// TwinCAT 3 PLC project Untitled1
// ProgramVersion: 3.1.4022.4
// libraries:
//   VisuElemBase, * (System)
//   VisuElems, * (System)
//   VisuElemsSpecialControls, * (System)
//   VisuElemsWinControls, * (System)
//   VisuInputs, * (System)
//   VisuNativeControl, * (System)
//   Tc2_FTP, * (Beckhoff Automation GmbH)
//   Tc2_MC2, * (Beckhoff Automation GmbH)
//   Tc2_NCI, * (Beckhoff Automation GmbH)
//   Tc2_Standard, * (Beckhoff Automation GmbH)
//   Tc2_System, * (Beckhoff Automation GmbH)
//   Tc2_Utilities, * (Beckhoff Automation GmbH)
//   Tc3_IotBase, * (Beckhoff Automation GmbH)
//   Tc3_JsonXml, * (Beckhoff Automation GmbH)
//   Tc3_Module, * (Beckhoff Automation GmbH)
//   VisuElemsDateTime Interfaces,newest,Intern
// project tree:
//   / GlobalTextList.TcGTLO, PlcTask.TcTTO, Visualization Manager.TcVMO (not stored)
//   GVLs/ COM.TcGVL, GVL.TcGVL
//   POUs/ ERROR.TcPOU, FTP.TcPOU, INIT.TcPOU, MAIN.TcPOU, POSITION.TcPOU, submqtt.TcPOU (not stored), commandDecoder.TcPOU
//   VISUs/ goPositionAbs.TcVIS, goPositionRel.TcVIS, Homing.TcVIS, Basic.TcVIS
// real-time tasks:
//   TASK PlcTask: cycle T#10ms, priority 20, ADS port 350
// motion (NC):
//   TASK NC-Task 1 SAF: cycle T#2ms, priority 4, ADS port 501
//   TASK NC-Task 1 SVB: cycle T#10ms, priority 8, ADS port 511
//   AXIS Axis X1 (id 1)
//     OtherSettings: AllowMotionCmdToSlave=true
//     encoder EncType=4
//       EncPara: ScaleFactorNumerator=40, ScaleFactorDenominator=12800, Inverse=true, MaxCount=#x0000ffff
//         SoftEndMinControl: Enable=true
//         SoftEndMaxControl: Enable=true, Range=275
//         Inc: RefSearchInverse=true, RefSyncInverse=false, RefMode=1, RefSoftSyncMask=#x0000ffff
//     drive DrvType=24
//       DrvPara: Inverse=true
//         Analog: VeloReferenz=400, ScaleFactorActTorque=0.1
//         TimeComp: TaskDelayCycles=1
//     controller CtrType=1
//       CtrPara: PriorControlFactor=1
//         PID: PosKp=25
//         Observer: BandWidth=20
//   AXIS Axis X2 (id 2)
//     OtherSettings: AllowMotionCmdToSlave=true
//     encoder EncType=4
//       EncPara: ScaleFactorNumerator=40, ScaleFactorDenominator=12800, Inverse=true, MaxCount=#x0000ffff
//         Inc: RefSoftSyncMask=#x0000ffff
//     drive DrvType=24
//       DrvPara: Inverse=true
//         Analog: VeloReferenz=400, ScaleFactorActTorque=0.1
//         TimeComp: TaskDelayCycles=1
//     controller CtrType=1
//       CtrPara: PriorControlFactor=1
//         PID: PosKp=25
//         Observer: BandWidth=20
//   AXIS Axis Y (id 4)
//     OtherSettings: AllowMotionCmdToSlave=true
//     encoder EncType=4
//       EncPara: ScaleFactorNumerator=40, ScaleFactorDenominator=12800, Inverse=true, MaxCount=#x0000ffff
//         SoftEndMinControl: Enable=true
//         SoftEndMaxControl: Enable=true, Range=275
//         Inc: RefSearchInverse=true, RefSyncInverse=false, RefMode=1, RefSoftSyncMask=#x0000ffff
//     drive DrvType=24
//       DrvPara: Inverse=true
//         Analog: VeloReferenz=400, ScaleFactorActTorque=0.1
//         TimeComp: TaskDelayCycles=1
//     controller CtrType=1
//       CtrPara: PriorControlFactor=1
//         PID: PosKp=25
//         Observer: BandWidth=20
//   AXIS Axis Z (id 3)
//     Velo: SlowManual=2, FastManual=5
//     OtherSettings: AllowMotionCmdToSlave=true
//     encoder EncType=4
//       EncPara: ScaleFactorNumerator=1, ScaleFactorDenominator=12800, MaxCount=#x0000ffff
//         Inc: RefSoftSyncMask=#x0000ffff
//     drive DrvType=24
//       Analog: VeloReferenz=10, ScaleFactorActTorque=0.1
//       TimeComp: TaskDelayCycles=1
//     controller CtrType=1
//       CtrPara: PriorControlFactor=1
//         PID: PosKp=25
//         Observer: BandWidth=20
// I/O:
//   DEVICE Device 3 (EtherCAT), AmsNetId 10.86.134.48.4.1
//     Term 1 (EK1100) [EK1100 EtherCAT Coupler (2A E-Bus)]
//       Term 2 (EL7031-0030) [EL7031-0030 1Ch. Stepper motor output stage (24V, 2.8A)]
//       Term 3 (EL7031-0030) [EL7031-0030 1Ch. Stepper motor output stage (24V, 2.8A)]
//       Term 4 (EL7031-0030) [EL7031-0030 1Ch. Stepper motor output stage (24V, 2.8A)]
//       Term 5 (EL7031-0030) [EL7031-0030 1Ch. Stepper motor output stage (24V, 2.8A)]
//       Term 6 (EL1008) [EL1008 8Ch. Dig. Input 24V, 3ms]
//       Term 7 (EL9011) [EL9011 End Terminal]
// variable links:
//   NC-Task 1 SAF/Axes/Axis X1 <-> Device 3 (EtherCAT)/Term 1 (EK1100)/Term 2 (EL7031-0030)
//     Drive/Inputs/In/nState1 @bit 3 <-> STM Status/Status/Error
//     Drive/Inputs/In/nState1 @bit 5 <-> STM Status/Status/Moving negative
//     Drive/Inputs/In/nState1 @bit 4 <-> STM Status/Status/Moving positive
//     Drive/Inputs/In/nState1 @bit 1 <-> STM Status/Status/Ready
//     Drive/Inputs/In/nState1 <-> STM Status/Status/Ready to enable
//     Drive/Inputs/In/nState1 @bit 6 <-> STM Status/Status/Torque reduced
//     Drive/Inputs/In/nState1 @bit 2 <-> STM Status/Status/Warning
//     Drive/Inputs/In/nState2 @bit 3 <-> STM Status/Status/Digital input 1
//     Drive/Inputs/In/nState2 @bit 4 <-> STM Status/Status/Digital input 2
//     Drive/Inputs/In/nState2 @bit 5 <-> STM Status/Status/Sync error
//     Drive/Inputs/In/nState2 @bit 7 <-> STM Status/Status/TxPDO Toggle
//     Drive/Inputs/In/nState4 @bit 1 <-> WcState/InputToggle
//     Drive/Inputs/In/nState4 <-> WcState/WcState
//     Drive/Outputs/Out/nCtrl1 <-> STM Control/Control/Enable
//     Drive/Outputs/Out/nCtrl1 @bit 2 <-> STM Control/Control/Reduce torque
//     Drive/Outputs/Out/nCtrl1 @bit 1 <-> STM Control/Control/Reset
//     Drive/Outputs/Out/nDataOut2[0] <-> STM Velocity/Velocity
//     Enc/Inputs/In/nDataIn1[0] <-> ENC Status compact/Counter value
//     Enc/Inputs/In/nDataIn2[0] <-> ENC Status compact/Latch value
//     Enc/Inputs/In/nState1 @bit 4 <-> ENC Status compact/Status/Counter overflow
//     Enc/Inputs/In/nState1 @bit 3 <-> ENC Status compact/Status/Counter underflow
//     Enc/Inputs/In/nState1 @bit 1 <-> ENC Status compact/Status/Latch extern valid
//     Enc/Inputs/In/nState1 @bit 2 <-> ENC Status compact/Status/Set counter done
//     Enc/Inputs/In/nState2 @bit 4 <-> ENC Status compact/Status/Status of extern latch
//     Enc/Inputs/In/nState2 @bit 5 <-> ENC Status compact/Status/Sync error
//     Enc/Inputs/In/nState2 @bit 7 <-> ENC Status compact/Status/TxPDO Toggle
//     Enc/Inputs/In/nState4 @bit 1 <-> WcState/InputToggle
//     Enc/Inputs/In/nState4 <-> WcState/WcState
//     Enc/Outputs/Out/nCtrl1 @bit 3 <-> ENC Control compact/Control/Enable latch extern on negative edge
//     Enc/Outputs/Out/nCtrl1 @bit 1 <-> ENC Control compact/Control/Enable latch extern on positive edge
//     Enc/Outputs/Out/nCtrl1 @bit 2 <-> ENC Control compact/Control/Set counter
//     Enc/Outputs/Out/nDataOut1[0] <-> ENC Control compact/Set counter value
//   NC-Task 1 SAF/Axes/Axis X2 <-> Device 3 (EtherCAT)/Term 1 (EK1100)/Term 3 (EL7031-0030)
//     Drive/Inputs/In/nState1 @bit 3 <-> STM Status/Status/Error
//     Drive/Inputs/In/nState1 @bit 5 <-> STM Status/Status/Moving negative
//     Drive/Inputs/In/nState1 @bit 4 <-> STM Status/Status/Moving positive
//     Drive/Inputs/In/nState1 @bit 1 <-> STM Status/Status/Ready
//     Drive/Inputs/In/nState1 <-> STM Status/Status/Ready to enable
//     Drive/Inputs/In/nState1 @bit 6 <-> STM Status/Status/Torque reduced
//     Drive/Inputs/In/nState1 @bit 2 <-> STM Status/Status/Warning
//     Drive/Inputs/In/nState2 @bit 3 <-> STM Status/Status/Digital input 1
//     Drive/Inputs/In/nState2 @bit 4 <-> STM Status/Status/Digital input 2
//     Drive/Inputs/In/nState2 @bit 5 <-> STM Status/Status/Sync error
//     Drive/Inputs/In/nState2 @bit 7 <-> STM Status/Status/TxPDO Toggle
//     Drive/Inputs/In/nState4 @bit 1 <-> WcState/InputToggle
//     Drive/Inputs/In/nState4 <-> WcState/WcState
//     Drive/Outputs/Out/nCtrl1 <-> STM Control/Control/Enable
//     Drive/Outputs/Out/nCtrl1 @bit 2 <-> STM Control/Control/Reduce torque
//     Drive/Outputs/Out/nCtrl1 @bit 1 <-> STM Control/Control/Reset
//     Drive/Outputs/Out/nDataOut2[0] <-> STM Velocity/Velocity
//     Enc/Inputs/In/nDataIn1[0] <-> ENC Status compact/Counter value
//     Enc/Inputs/In/nDataIn2[0] <-> ENC Status compact/Latch value
//     Enc/Inputs/In/nState1 @bit 4 <-> ENC Status compact/Status/Counter overflow
//     Enc/Inputs/In/nState1 @bit 3 <-> ENC Status compact/Status/Counter underflow
//     Enc/Inputs/In/nState1 @bit 1 <-> ENC Status compact/Status/Latch extern valid
//     Enc/Inputs/In/nState1 @bit 2 <-> ENC Status compact/Status/Set counter done
//     Enc/Inputs/In/nState2 @bit 4 <-> ENC Status compact/Status/Status of extern latch
//     Enc/Inputs/In/nState2 @bit 5 <-> ENC Status compact/Status/Sync error
//     Enc/Inputs/In/nState2 @bit 7 <-> ENC Status compact/Status/TxPDO Toggle
//     Enc/Inputs/In/nState4 @bit 1 <-> WcState/InputToggle
//     Enc/Inputs/In/nState4 <-> WcState/WcState
//     Enc/Outputs/Out/nCtrl1 @bit 3 <-> ENC Control compact/Control/Enable latch extern on negative edge
//     Enc/Outputs/Out/nCtrl1 @bit 1 <-> ENC Control compact/Control/Enable latch extern on positive edge
//     Enc/Outputs/Out/nCtrl1 @bit 2 <-> ENC Control compact/Control/Set counter
//     Enc/Outputs/Out/nDataOut1[0] <-> ENC Control compact/Set counter value
//   NC-Task 1 SAF/Axes/Axis Y <-> Device 3 (EtherCAT)/Term 1 (EK1100)/Term 5 (EL7031-0030)
//     Drive/Inputs/In/nState1 @bit 3 <-> STM Status/Status/Error
//     Drive/Inputs/In/nState1 @bit 5 <-> STM Status/Status/Moving negative
//     Drive/Inputs/In/nState1 @bit 4 <-> STM Status/Status/Moving positive
//     Drive/Inputs/In/nState1 @bit 1 <-> STM Status/Status/Ready
//     Drive/Inputs/In/nState1 <-> STM Status/Status/Ready to enable
//     Drive/Inputs/In/nState1 @bit 6 <-> STM Status/Status/Torque reduced
//     Drive/Inputs/In/nState1 @bit 2 <-> STM Status/Status/Warning
//     Drive/Inputs/In/nState2 @bit 3 <-> STM Status/Status/Digital input 1
//     Drive/Inputs/In/nState2 @bit 4 <-> STM Status/Status/Digital input 2
//     Drive/Inputs/In/nState2 @bit 5 <-> STM Status/Status/Sync error
//     Drive/Inputs/In/nState2 @bit 7 <-> STM Status/Status/TxPDO Toggle
//     Drive/Inputs/In/nState4 @bit 1 <-> WcState/InputToggle
//     Drive/Inputs/In/nState4 <-> WcState/WcState
//     Drive/Outputs/Out/nCtrl1 <-> STM Control/Control/Enable
//     Drive/Outputs/Out/nCtrl1 @bit 2 <-> STM Control/Control/Reduce torque
//     Drive/Outputs/Out/nCtrl1 @bit 1 <-> STM Control/Control/Reset
//     Drive/Outputs/Out/nDataOut2[0] <-> STM Velocity/Velocity
//     Enc/Inputs/In/nDataIn1[0] <-> ENC Status compact/Counter value
//     Enc/Inputs/In/nDataIn2[0] <-> ENC Status compact/Latch value
//     Enc/Inputs/In/nState1 @bit 4 <-> ENC Status compact/Status/Counter overflow
//     Enc/Inputs/In/nState1 @bit 3 <-> ENC Status compact/Status/Counter underflow
//     Enc/Inputs/In/nState1 @bit 1 <-> ENC Status compact/Status/Latch extern valid
//     Enc/Inputs/In/nState1 @bit 2 <-> ENC Status compact/Status/Set counter done
//     Enc/Inputs/In/nState2 @bit 4 <-> ENC Status compact/Status/Status of extern latch
//     Enc/Inputs/In/nState2 @bit 5 <-> ENC Status compact/Status/Sync error
//     Enc/Inputs/In/nState2 @bit 7 <-> ENC Status compact/Status/TxPDO Toggle
//     Enc/Inputs/In/nState4 @bit 1 <-> WcState/InputToggle
//     Enc/Inputs/In/nState4 <-> WcState/WcState
//     Enc/Outputs/Out/nCtrl1 @bit 3 <-> ENC Control compact/Control/Enable latch extern on negative edge
//     Enc/Outputs/Out/nCtrl1 @bit 1 <-> ENC Control compact/Control/Enable latch extern on positive edge
//     Enc/Outputs/Out/nCtrl1 @bit 2 <-> ENC Control compact/Control/Set counter
//     Enc/Outputs/Out/nDataOut1[0] <-> ENC Control compact/Set counter value
//   NC-Task 1 SAF/Axes/Axis Z <-> Device 3 (EtherCAT)/Term 1 (EK1100)/Term 4 (EL7031-0030)
//     Drive/Inputs/In/nState1 @bit 3 <-> STM Status/Status/Error
//     Drive/Inputs/In/nState1 @bit 5 <-> STM Status/Status/Moving negative
//     Drive/Inputs/In/nState1 @bit 4 <-> STM Status/Status/Moving positive
//     Drive/Inputs/In/nState1 @bit 1 <-> STM Status/Status/Ready
//     Drive/Inputs/In/nState1 <-> STM Status/Status/Ready to enable
//     Drive/Inputs/In/nState1 @bit 6 <-> STM Status/Status/Torque reduced
//     Drive/Inputs/In/nState1 @bit 2 <-> STM Status/Status/Warning
//     Drive/Inputs/In/nState2 @bit 3 <-> STM Status/Status/Digital input 1
//     Drive/Inputs/In/nState2 @bit 4 <-> STM Status/Status/Digital input 2
//     Drive/Inputs/In/nState2 @bit 5 <-> STM Status/Status/Sync error
//     Drive/Inputs/In/nState2 @bit 7 <-> STM Status/Status/TxPDO Toggle
//     Drive/Inputs/In/nState4 @bit 1 <-> WcState/InputToggle
//     Drive/Inputs/In/nState4 <-> WcState/WcState
//     Drive/Outputs/Out/nCtrl1 <-> STM Control/Control/Enable
//     Drive/Outputs/Out/nCtrl1 @bit 2 <-> STM Control/Control/Reduce torque
//     Drive/Outputs/Out/nCtrl1 @bit 1 <-> STM Control/Control/Reset
//     Drive/Outputs/Out/nDataOut2[0] <-> STM Velocity/Velocity
//     Enc/Inputs/In/nDataIn1[0] <-> ENC Status compact/Counter value
//     Enc/Inputs/In/nDataIn2[0] <-> ENC Status compact/Latch value
//     Enc/Inputs/In/nState1 @bit 4 <-> ENC Status compact/Status/Counter overflow
//     Enc/Inputs/In/nState1 @bit 3 <-> ENC Status compact/Status/Counter underflow
//     Enc/Inputs/In/nState1 @bit 1 <-> ENC Status compact/Status/Latch extern valid
//     Enc/Inputs/In/nState1 @bit 2 <-> ENC Status compact/Status/Set counter done
//     Enc/Inputs/In/nState2 @bit 4 <-> ENC Status compact/Status/Status of extern latch
//     Enc/Inputs/In/nState2 @bit 5 <-> ENC Status compact/Status/Sync error
//     Enc/Inputs/In/nState2 @bit 7 <-> ENC Status compact/Status/TxPDO Toggle
//     Enc/Inputs/In/nState4 @bit 1 <-> WcState/InputToggle
//     Enc/Inputs/In/nState4 <-> WcState/WcState
//     Enc/Outputs/Out/nCtrl1 @bit 3 <-> ENC Control compact/Control/Enable latch extern on negative edge
//     Enc/Outputs/Out/nCtrl1 @bit 1 <-> ENC Control compact/Control/Enable latch extern on positive edge
//     Enc/Outputs/Out/nCtrl1 @bit 2 <-> ENC Control compact/Control/Set counter
//     Enc/Outputs/Out/nDataOut1[0] <-> ENC Control compact/Set counter value
//   Untitled1/Untitled1 Instance <-> Device 3 (EtherCAT)/Term 1 (EK1100)/Term 6 (EL1008)
//     PlcTask Inputs/GVL.bX1 <-> Channel 3/Input
//     PlcTask Inputs/GVL.bX2 <-> Channel 4/Input
//     PlcTask Inputs/GVL.bY1 <-> Channel 1/Input
//     PlcTask Inputs/GVL.bY2 <-> Channel 2/Input
//   Untitled1/Untitled1 Instance <-> NC-Task 1 SAF/Axes/Axis X1
//     PlcTask Inputs/GVL.As_Xa.NcToPlc <-> Outputs/ToPlc
//     PlcTask Outputs/GVL.As_Xa.PlcToNc <-> Inputs/FromPlc
//   Untitled1/Untitled1 Instance <-> NC-Task 1 SAF/Axes/Axis X2
//     PlcTask Inputs/GVL.As_Xb.NcToPlc <-> Outputs/ToPlc
//     PlcTask Outputs/GVL.As_Xb.PlcToNc <-> Inputs/FromPlc
//   Untitled1/Untitled1 Instance <-> NC-Task 1 SAF/Axes/Axis Y
//     PlcTask Inputs/GVL.As_Y.NcToPlc <-> Outputs/ToPlc
//     PlcTask Outputs/GVL.As_Y.PlcToNc <-> Inputs/FromPlc
//   Untitled1/Untitled1 Instance <-> NC-Task 1 SAF/Axes/Axis Z
//     PlcTask Inputs/GVL.As_Z.NcToPlc <-> Outputs/ToPlc
//     PlcTask Outputs/GVL.As_Z.PlcToNc <-> Inputs/FromPlc
//   Untitled1/Untitled1 Instance <-> NC-Task 1 SAF/G-code
//     PlcTask Inputs/GVL.ChannelInput <-> Outputs/ToPlc
//     PlcTask Outputs/GVL.ChannelOutput <-> Inputs/FromPlc

CONFIGURATION Untitled1
    RESOURCE PLC ON TwinCAT3
        TASK PlcTask(INTERVAL := T#10ms, PRIORITY := 20);
        PROGRAM MAIN WITH PlcTask : MAIN;
    END_RESOURCE
END_CONFIGURATION

// ---- GVLs/COM.TcGVL
{attribute 'qualified_only'}
VAR_GLOBAL
	
	doHome : BOOL;
	
END_VAR

// ---- GVLs/GVL.TcGVL
{attribute 'qualified_only'}
VAR_GLOBAL
	As_Xa : AXIS_REF;
	As_Xb : AXIS_REF;
	As_Y : AXIS_REF;
	As_Z : AXIS_REF;
	
	ChannelInput AT %I* : NCTOPLC_NCICHANNEL_REF;
	ChannelOutput AT %Q* : PLCTONC_NCICHANNEL_REF;
	
	StopALL : bool;
	
	bX1 AT%I* : BOOL;
	bX2 AT%I* : BOOL;
	bY1 AT%I* : BOOL;
	bY2 AT%I* : BOOL;
	
	stReceivedData	: STRING(255);
	
	
END_VAR

// ---- POUs/MAIN.TcPOU
PROGRAM MAIN
VAR
	
END_VAR

//main program
INIT();

//SUBMQTT Connection and receiving
//submqtt();

//FTP
FTP();

//AT COmmands decoder
//commandDecoder();

//Get positions
POSITION();

//Error
ERROR();

END_PROGRAM

// ---- POUs/INIT.TcPOU
PROGRAM INIT
VAR
	MCPower_Xa : MC_Power;
	MCPower_Xb : MC_Power;
	MCPower_Y : MC_Power;
	MCPower_Z : MC_Power;
	
	MCResetXa: MC_Reset;
	MCResetXb: MC_Reset;
	MCResetY: MC_Reset;
	MCResetZ: MC_Reset;
	
	fb_MCGearIn: MC_GearIn;
	fb_MCGearOut: MC_GearOut;

	fb_MCHOME_X: MC_Home;
	fb_MCHOME_Y: MC_Home;

	bEN		: BOOL;
	bENCouple : BOOL;
	bReset	: BOOL;
	bGearIn : BOOL;
	bHome	: BOOL;
		
	fb_BuildGroup: CfgBuild3DGroup;
	fb_ReconfigGroup: CfgReconfigGroup;
	fb_LoadProg: ItpLoadProgEx;
	fb_StartStop: ItpStartStopEx;
	fb_Reset: ItpResetEx2;
	
	bBuildGroup: BOOL;
	bLoad: BOOL;
	bStart: BOOL;
	bStop: BOOL;
	
END_VAR

MCPower_Xa(
	Axis:= GVL.As_Xa, 
	Enable:= bENCouple OR bEN, 
	Enable_Positive:= bENCouple OR bEN, 
	Enable_Negative:= bENCouple OR bEN, 
	Override:= 100 );
	
MCPower_Xb(
	Axis:= GVL.As_Xb, 
	Enable:= bENCouple OR bEN, 
	Enable_Positive:= bENCouple OR bEN, 
	Enable_Negative:= bENCouple OR bEN, 
	Override:= 100 );
	
MCPower_Y(
	Axis:= GVL.As_Y, 
	Enable:= bENCouple OR bEN, 
	Enable_Positive:= bENCouple OR bEN, 
	Enable_Negative:= bENCouple OR bEN, 
	Override:= 100 );
	
MCPower_Z(
	Axis:= GVL.As_Z, 
	Enable:= bENCouple OR bEN, 
	Enable_Positive:= bENCouple OR bEN, 
	Enable_Negative:= bENCouple OR bEN, 
	Override:= 100 );
	
MCResetXa(
	Axis:= GVL.As_Xa, 
	Execute:= bReset );
	
MCResetXb(
	Axis:= GVL.As_Xb, 
	Execute:= bReset );

MCResetY(
	Axis:= GVL.As_Y, 
	Execute:= bReset );

MCResetZ(
	Axis:= GVL.As_Z, 
	Execute:= bReset );
	
fb_MCGearIn(
	Master:= GVL.As_Xa, 
	Slave:= GVL.As_Xb, 
	Execute:= bENCouple OR bGearIn, 
	RatioNumerator:= 1, 
	RatioDenominator:= 1 );
	
fb_MCGearOut(
	Slave:= GVL.As_Xb,
	Execute:= NOT(bENCouple OR bGearIn) );
	
fb_MCHOME_X(
	Axis:= GVL.As_Xa, 
	Execute:= ( bHome OR COM.doHome ) AND ( bENCouple OR bGearIn ), 
	Position:= 0, 
	bCalibrationCam:= GVL.bX1 );
	
fb_MCHOME_Y(
	Axis:= GVL.As_Y, 
	Execute:= ( bHome OR COM.doHome ) AND ( bENCouple OR bGearIn ), 
	Position:= 0, 
	bCalibrationCam:= GVL.bY1 );
	
NCI();

ACTION NCI:
fb_BuildGroup(
	bExecute:= bBuildGroup, 
	nGroupId:= GVL.ChannelInput.GrpId, 
	nXAxisId:= GVL.As_Xa.NcToPlc.AxisId, 
	nYAxisId:= GVL.As_Y.NcToPlc.AxisId, 
	nZAxisId:= GVL.As_Z.NcToPlc.AxisId, 
	tTimeOut:= T#1S );
	
fb_ReconfigGroup(
	bExecute:= NOT(bBuildGroup), 
	nGroupId:= GVL.ChannelInput.GrpId, 
	tTimeOut:= T#1S );
	
ItpSetOverridePercent(fOverridePercent:= 100, sPlcToNci:= GVL.ChannelOutput);

fb_LoadProg(
	sNciToPlc:= GVL.ChannelInput, 
	bExecute:= bLoad, 
	sPrg:= '\HARD DISK\TWINCAT\Mc\Nci\Gcode_test1.nc', 
	nLength:= LEN('\HARD DISK\TWINCAT\Mc\Nci\Gcode_test1.nc'), 
	tTimeOut:= T#1S );
	
fb_StartStop(
	bStart:= bStart, 
	bStop:= bStop, 
	tTimeOut:= T#1S, 
	sNciToPlc:= GVL.ChannelInput );
	
fb_Reset(
	bExecute:= bReset, 
	tTimeOut:= T#1S, 
	sNciToPlc:= GVL.ChannelInput );
END_ACTION

END_PROGRAM

// ---- POUs/POSITION.TcPOU
PROGRAM POSITION
VAR
	MoveRel_X : MC_MoveRelative;
	MoveRel_Y : MC_MoveRelative;
	MoveRel_Z : MC_MoveRelative;
	
	MoveAbs_X : MC_MoveAbsolute;
	MoveAbs_Y : MC_MoveAbsolute;
	MoveAbs_Z : MC_MoveAbsolute;
	
	SetZToZero 	: MC_SetPosition;
	SetZpos		: BOOL;
	
	DoRel_X : BOOL;
	DoRel_Y : BOOL;
	DoRel_Z : BOOL;
	
	DoAbs_X : BOOL;
	DoAbs_Y : BOOL;
	DoAbs_Z : BOOL;

	Busy : BOOL;
	Done : BOOL;
	
	abs_X : INT := 0;
	abs_Y : INT := 0;
	abs_Z : INT := 0;
	
	Rel_X : INT := 0;
	Rel_Y : INT := 0;
	Rel_Z : INT := 5;
	
	vel_X : INT := 200;
	vel_Y : INT := 200;
	vel_Z : INT := 3;
	
END_VAR

//jog 

IF(	MoveRel_X.Busy OR MoveAbs_X.Busy OR	MoveRel_Y.Busy OR MoveAbs_Y.Busy OR	MoveRel_Z.Busy OR MoveAbs_Z.Busy )THEN
	Busy := TRUE;
	Done := FALSE;
ELSE
	Busy := FALSE;
	Done := TRUE;
END_IF

//X			
MoveRel_X(Axis := GVL.As_Xa,	
		Execute := DoRel_X AND ( (INIT.bGearIn AND INIT.bEN) OR INIT.bENCouple ),
		Distance := Rel_X,
		Velocity := vel_X);
		
MoveAbs_X(Axis := GVL.As_Xa,
		Execute := DoAbs_X AND ( (INIT.bGearIn AND INIT.bEN) OR INIT.bENCouple ),
		Position := abs_X,
		Velocity := vel_X);
		
//Y
MoveRel_Y(Axis := GVL.As_Y,
		Execute := DoRel_Y AND (INIT.bEN OR INIT.bENCouple),
		Distance := Rel_Y,
		Velocity := vel_Y);
		
MoveAbs_Y(Axis := GVL.As_Y,
		Execute := DoAbs_Y AND (INIT.bEN OR INIT.bENCouple),
		Position := abs_Y,
		Velocity := vel_Y);

//Z
MoveRel_Z(Axis := GVL.As_Z,
		Execute := DoRel_Z AND (INIT.bEN OR INIT.bENCouple),
		Distance := Rel_Z,
		Velocity := vel_Z);
		
MoveAbs_Z(Axis := GVL.As_Z,
		Execute := DoAbs_Z AND (INIT.bEN OR INIT.bENCouple),
		Position := abs_Z,
		Velocity := vel_Z);
		
//set Z postition to zero
SetZToZero(Axis := GVL.As_Z, 
			Execute := SetZpos,
			Position := 0, 
			Mode := FALSE);

END_PROGRAM

// ---- POUs/FTP.TcPOU
PROGRAM FTP
VAR
END_VAR

//https://download.beckhoff.com/download/document/automation/twincat3/TF6300_TC3_FTP_CLIENT_EN.pdf

END_PROGRAM

// ---- POUs/ERROR.TcPOU
PROGRAM ERROR
VAR
	StopX_a : MC_Stop;
	StopX_b : MC_Stop;
	StopY : MC_Stop;
	StopZ : MC_Stop;

END_VAR

// https://infosys.beckhoff.com/english.php?content=../content/1033/tccncmcplatform_fb/html/mcstop.htm&id=
// start stop pause continue

StopX_a(Axis := gvl.As_Xa,
		Execute := GVL.StopALL);

StopX_b(Axis := gvl.As_Xb,
		Execute := GVL.StopALL);

StopY(Axis := gvl.As_Y,
		Execute := GVL.StopALL);
		
StopZ(Axis := gvl.As_Z,
		Execute := GVL.StopALL);

END_PROGRAM

// ---- POUs/commandDecoder.TcPOU

PROGRAM commandDecoder
VAR
	Command : STRING;
	Head_Loaded : STRING;
	Coordinate : WORD;
END_VAR

Command := F_ToLCase(GVL.stReceivedData);
GVL.stReceivedData := '';

//example
IF(Command = 'start') THEN
	Command := '';
	
ELSIF(Command = 'stop') THEN
	COM.doHome := FALSE;
	Command := '';
	
ELSIF(Command = 'home') THEN
	COM.doHome := TRUE;
	Command := '';
		
ELSE
	COM.doHome := FALSE; //temp
	Command := '';
	
END_IF;

END_PROGRAM

// ---- GlobalTextList.TcGTLO
TEXTLIST GlobalTextList
  943 = 'Absolute'
  163 = 'Couple'
  730 = 'Group'
  610 = 'Home'
  23 = 'Load'
  172 = 'move abs X'
  424 = 'Move abs X'
  68 = 'move abs Y'
  700 = 'Move abs Y'
  459 = 'move ABS z'
  52 = 'move abs z'
  760 = 'move abs Z'
  258 = 'Move abs Z'
  193 = 'move rel X'
  135 = 'Move rel X'
  829 = 'move rel Y'
  787 = 'Move rel Y'
  698 = 'move rel z'
  917 = 'move rel Z'
  750 = 'Move rel z'
  793 = 'Niet gebruiken'
  769 = 'Reconfig'
  653 = 'Relative'
  187 = 'Reset'
  285 = 'set z on pos 0'
  244 = 'Set Z pos to 0'
  127 = 'Start'
  887 = 'Stop'
  966 = 'STOP'
END_TEXTLIST

// ---- VISUs/goPositionAbs.TcVIS
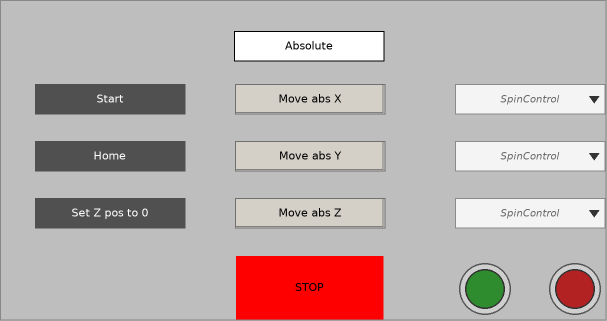
VISUALIZATION goPositionAbs  // 607x321
    Button (235,84 150x30), "Move abs X"
        tap POSITION.DoAbs_X
    Button (235,141 150x30), "Move abs Y"
        tap POSITION.DoAbs_Y
    Button (235,198 150x30), "Move abs Z"
        tap POSITION.DoAbs_Z
    Rectangle (35,141 150x30), "Home"
        tap INIT.bHome
    Rectangle (35,84 150x30), "Start", colour toggle: INIT.bENCouple
        toggle INIT.bENCouple
    Rectangle (35,198 150x30), "Set Z pos to 0"
        tap POSITION.SetZpos
    SpinControl (455,84 150x30), variable: POSITION.abs_X
        OnMouseDown: write POSITION.abs_X via Edit, min 0, max 275
    SpinControl (455,141 150x30), variable: POSITION.abs_Y
        OnMouseDown: write POSITION.abs_Y via Edit, min 0, max 275
    SpinControl (455,198 150x30), variable: POSITION.abs_Z
        OnMouseDown: write POSITION.abs_Z via Edit, min 0, max 90
    Rectangle (236,256 147x63), "STOP", colour toggle: GVL.StopALL
        toggle GVL.StopALL
    Lamp1 (455,259 60x60), variable: POSITION.Done, style: Lamp-Lamp1-Green
    Lamp1 (545,259 60x60), variable: POSITION.Busy, style: Lamp-Lamp1-Red
    Rectangle (234,31 150x30), "Absolute"
END_VISUALIZATION

// ---- VISUs/goPositionRel.TcVIS
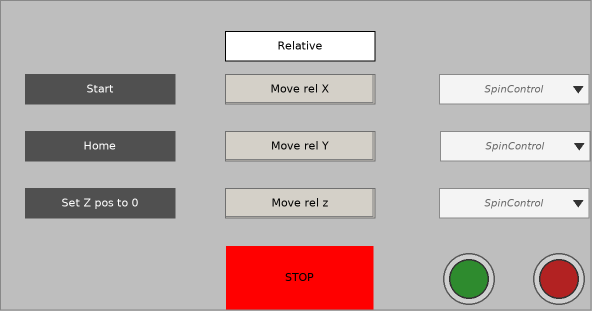
VISUALIZATION goPositionRel  // 592x311
    Button (225,74 150x30), "Move rel X"
        tap POSITION.DoRel_X
    Button (225,131 150x30), "Move rel Y"
        tap POSITION.DoRel_Y
    Button (225,188 150x30), "Move rel z"
        tap POSITION.DoRel_Z
    Rectangle (226,246 147x63), "STOP", colour toggle: GVL.StopALL
        toggle GVL.StopALL
    Rectangle (25,131 150x30), "Home"
        tap INIT.bHome
    Rectangle (25,74 150x30), "Start", colour toggle: INIT.bENCouple
        toggle INIT.bENCouple
    Rectangle (25,188 150x30), "Set Z pos to 0"
        tap POSITION.SetZpos
    SpinControl (439,74 150x30), variable: POSITION.Rel_X
        OnMouseDown: write POSITION.Rel_X via Edit, min 0, max 300
    SpinControl (440,131 150x30), variable: POSITION.Rel_Y
        OnMouseDown: write POSITION.Rel_Y via Edit, min 0, max 300
    SpinControl (439,188 150x30), variable: POSITION.Rel_Z
        OnMouseDown: write POSITION.Rel_Z via Edit, min -80, max 80
    Lamp1 (439,249 60x60), variable: POSITION.Done, style: Lamp-Lamp1-Green
    Lamp1 (529,249 60x60), variable: POSITION.Busy, style: Lamp-Lamp1-Red
    Rectangle (225,31 150x30), "Relative"
END_VISUALIZATION

// ---- VISUs/Homing.TcVIS
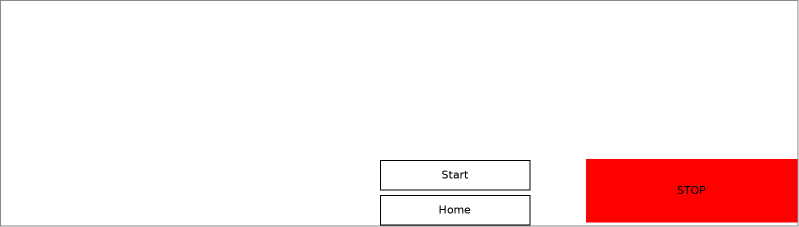
VISUALIZATION Homing  // 799x227
    Rectangle (380,195 150x30), "Home"
        tap INIT.bHome
    Rectangle (380,160 150x30), "Start", colour toggle: INIT.bEN
        toggle INIT.bENCouple
    Rectangle (586,159 211x63), "STOP", colour toggle: GVL.StopALL
        toggle GVL.StopALL
END_VISUALIZATION

// ---- VISUs/Basic.TcVIS
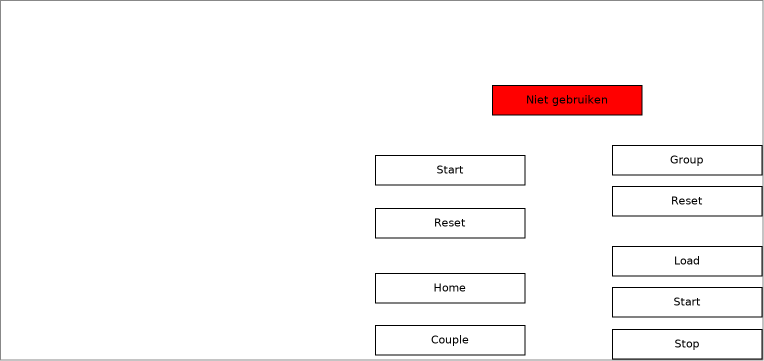
VISUALIZATION Basic  // 764x361
    Rectangle (375,325 150x30), "Couple", colour toggle: INIT.bGearIn
        toggle INIT.bGearIn
    Rectangle (375,273 150x30), "Home"
        tap INIT.bHome
    Rectangle (375,155 150x30), "Start", colour toggle: INIT.bEN
        toggle INIT.bEN
    Rectangle (375,208 150x30), "Reset", colour toggle: INIT.bReset
        tap INIT.bReset
    Rectangle (612,145 150x30), "Group", colour toggle: POU_NCI.bBuildGroup
        toggle POU_NCI.bBuildGroup
    Rectangle (612,186 150x30), "Reset"
        tap POU_NCI.bReset
    Rectangle (612,287 150x30), "Start"
        tap POU_NCI.bStart
    Rectangle (612,329 150x30), "Stop"
        tap POU_NCI.bStop
    Rectangle (612,246 150x30), "Load"
        tap POU_NCI.bLoad
    Rectangle (492,85 150x30), "Niet gebruiken"
END_VISUALIZATION
